FUNCTION_BLOCK SPLIT_AL_INTO_AD (* this Function splits the 2 AD (DWORD) adapters from a AL (LWORD) *)
  (* Standard: 61499-2; Description: Copyright (c) 2026 Meisterschulen am Ostbahnhof SPDX-License-Identifier: EPL-2.0 *)
  (* Version 1.0, 2026-05-16, Franz Höpfinger, Meisterschulen am Ostbahnhof, initial API and implementation and/or initial documentation *)
  PACKAGE adapter::splitting;
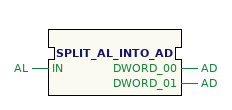
  SOCKETS
    IN : adapter::types::unidirectional::AL; (* LWORD Input *)
  END_SOCKETS
  PLUGS
    DWORD_00 : adapter::types::unidirectional::AD; (* DWord 0 *)
    DWORD_01 : adapter::types::unidirectional::AD; (* DWord 1 *)
  END_PLUGS
END_FUNCTION_BLOCK
